{attribute addProperty BoxType "KL9900-0064"}
{attribute addProperty Id "Key_1AT %I*BOOL000Key_2AT %I*BOOL000Key_3AT %I*BOOL000Key_4AT %I*BOOL000Input_1AT %I*BOOL000Input_2AT %I*BOOL000Input_3AT %I*BOOL000Input_4AT %I*BOOL000LED_1AT %Q*BOOL000LED_2AT %Q*BOOL000LED_3AT %Q*BOOL000LED_4AT %Q*BOOL000"}
{attribute addProperty CRC "2070896559"}
{attribute addProperty SizeInBites "0"}
{attribute addProperty SizeInBytes "0"}
TYPE Channel_7B6F5FAF :
STRUCT
	{attribute addProperty Name "Key_1"}
	Key_1 AT %I* : BOOL;
	{attribute addProperty Name "Key_2"}
	Key_2 AT %I* : BOOL;
	{attribute addProperty Name "Key_3"}
	Key_3 AT %I* : BOOL;
	{attribute addProperty Name "Key_4"}
	Key_4 AT %I* : BOOL;
	{attribute addProperty Name "Input_1"}
	Input_1 AT %I* : BOOL;
	{attribute addProperty Name "Input_2"}
	Input_2 AT %I* : BOOL;
	{attribute addProperty Name "Input_3"}
	Input_3 AT %I* : BOOL;
	{attribute addProperty Name "Input_4"}
	Input_4 AT %I* : BOOL;
	{attribute addProperty Name "LED_1"}
	LED_1 AT %Q* : BOOL;
	{attribute addProperty Name "LED_2"}
	LED_2 AT %Q* : BOOL;
	{attribute addProperty Name "LED_3"}
	LED_3 AT %Q* : BOOL;
	{attribute addProperty Name "LED_4"}
	LED_4 AT %Q* : BOOL;
END_STRUCT
END_TYPE

(* stored: Version 1.2.0.0, ProductVersion 3.1.4024.9
   DUT Channel_7B6F5FAF: Id {3ebe101a-bb83-485a-99bd-b28942c22437} *)
